// TwinCAT 3 PLC project XMLServerTesten
// ProgramVersion: 3.1.4023.0
// libraries:
//   Tc2_Standard, * (Beckhoff Automation GmbH)
//   Tc2_System, * (Beckhoff Automation GmbH)
//   Tc2_Utilities, * (Beckhoff Automation GmbH)
//   Tc2_XmlDataSrv, * (Beckhoff Automation GmbH)
//   Tc3_Module, * (Beckhoff Automation GmbH)
// project tree:
//   DUTs/ st_Datensatz.TcDUT, ST_TimeDiff.TcDUT (not stored), XMLHeader.TcDUT
//   / PlcTask.TcTTO (not stored)
//   POUs/ Get_Diff.TcPOU, fileT_to_sysT.TcPOU (not stored), MAIN.TcPOU, POU.TcPOU, RecordEndTime.TcPOU, RecordStartTime.TcPOU, write_to_Buffer.TcPOU, write_to_XML.TcPOU, XMLTesten.TcPOU

// ---- DUTs/st_Datensatz.TcDUT
TYPE st_Datensatz :
STRUCT
	Timestamp : STRING ;
	roomnum : REAL;
	temp : REAL;
	signal3 : REAL;
	signal4 : REAL;
	signal5 : REAL;
	signal6 : REAL;
	signal7 : REAL;
	signal8 : REAL;
END_STRUCT
END_TYPE

// ---- DUTs/XMLHeader.TcDUT
TYPE XMLHeader :
STRUCT
	MaschineNummer : STRING:= '1234567890';
	Manufacturer : STRING := 'Beckhoff';
	Maschinetype : STRING:= 'cx2040.1.1.1';
	Customer : STRING:= 'liyizhen23333';
	WriteTimeDiff : ST_TimeDiff;
END_STRUCT
END_TYPE

// ---- POUs/Get_Diff.TcPOU
FUNCTION_BLOCK Get_Diff
VAR_INPUT
	BeginLo: UDINT;
	BeginHi: UDINT;
	EndLo: UDINT;
	EndHi: UDINT;
END_VAR
VAR_OUTPUT
	WriteTimeDiff: ST_TimeDiff;
END_VAR
VAR
	HiDiff : UDINT;
	LoDiff : UDINT;
	SysTime : TIMESTRUCT;
	SysTimeBegin: TIMESTRUCT;
	SysTimeFinish: TIMESTRUCT;
	fileT_to_sysT_Begin: fileT_to_sysT;
	fileT_to_sysT_Finish: fileT_to_sysT;
END_VAR

HiDiff := EndHi - BeginHi;
LoDiff := EndLo - BeginLo;

//change hex time to hh:mm:ss time
fileT_to_sysT_Begin(T_LoDW := LoDiff, T_HiDW := HiDiff);
SysTime := fileT_to_sysT_Begin.sysT;

WriteTimeDiff.mMillisecond:= SysTime.wMilliseconds;
WriteTimeDiff.sSecond:= SysTime.wSecond;

END_FUNCTION_BLOCK

// ---- POUs/MAIN.TcPOU
PROGRAM MAIN
VAR
	XMLTesten : XMLTesten;
END_VAR

XMLTesten();

END_PROGRAM

// ---- POUs/XMLTesten.TcPOU
FUNCTION_BLOCK XMLTesten
VAR_INPUT
END_VAR
VAR_OUTPUT
END_VAR
VAR
	bFinish : BOOL;
	RecordStartTime : RecordStartTime;
	write_to_Buffer : write_to_Buffer;
	RecordEndTime : RecordEndTime;
	write_to_XML : write_to_XML;
	get_Diff : get_Diff;
	
	Buffer : ARRAY[1..100] OF st_Datensatz;
	m: INT :=1;
	StopRecordStart: BOOL := TRUE;
	DownTrigDetect: F_TRIG;
	WriteTimeDiff: ST_TimeDiff;
END_VAR

//record the start timestamp of writing to buffer
IF StopRecordStart THEN
	RecordStartTime(StartFlag := TRUE);
END_IF
StopRecordStart := FALSE; 			//be set so that the start timestamp is not refreshed when writing datensatz2

//when recordstarttime is finished the datensatz is written
IF RecordStartTime.RecordStFinish THEN
	write_to_Buffer(m := m,startrecord := TRUE);
	Buffer[m]:= write_to_Buffer.Datensatz;
	m :=m+1;
END_IF

//when 100 datensatz are written in buffer, record the end timestamp
IF m = 101 THEN
	RecordEndTime(EndFlag := TRUE);
	bFinish :=TRUE;
	m :=102;
END_IF

IF m = 110 THEN
	m := 1;
END_IF

//get timeintervall for writing into buffer (10ms*n)
get_Diff(WriteTimeDiff=>WriteTimeDiff,BeginLo := RecordStartTime.BeginLo,BeginHi := RecordStartTime.BeginHi,EndLo := RecordEndTime.EndLo, EndHi := RecordEndTime.EndHi);

//write data from buffer to xml file
IF bFinish THEN
	write_to_XML(WriteTimeDiffHeader := WriteTimeDiff,LogInput := Buffer,bExecute := TRUE);
END_IF

END_FUNCTION_BLOCK

// ---- POUs/RecordStartTime.TcPOU
FUNCTION_BLOCK RecordStartTime
VAR_INPUT
	StartFlag: BOOL := FALSE;
END_VAR
VAR_OUTPUT
	RecordStFinish : BOOL :=FALSE;
	BeginLo: UDINT;
	BeginHi: UDINT;
END_VAR
VAR
	UpTrigDetect: R_TRIG;
	MyTimer: getsystemtime;
	Delay: TON;
END_VAR

//start to get system time
MyTimer();

//detect the trigger: false to true
UpTrigDetect(CLK:=StartFlag);

//record beginning Timestamp of initializing period
IF UpTrigDetect.Q THEN
	BeginLo := MyTimer.timeLoDW;								
	BeginHi := MyTimer.timeHiDW;
END_IF

RecordStFinish := TRUE;

//time to wait before next cycle

Delay(IN := TRUE, PT := T#5S);            
IF NOT(Delay.Q) THEN
	RETURN;
END_IF
Delay.IN := FALSE;

END_FUNCTION_BLOCK

// ---- POUs/write_to_Buffer.TcPOU
FUNCTION_BLOCK write_to_Buffer
VAR_INPUT
	startrecord : BOOL;
END_VAR
VAR_OUTPUT
	Datensatz : st_Datensatz;
END_VAR
VAR
	GetTime : NT_GetTime;
	GETTIMESTART : BOOL :=TRUE;
	Timestamp : T_Filetime;
	MyTimer: getsystemtime;
	TimestampSYS: TIMESTRUCT;
END_VAR

//100 values in array
	//GetTime(START := GETTIMESTART,TIMESTR => Timestamp);
	//Datensatz.Timestamp := SYSTEMTIME_TO_STRING(Timestamp);
	MyTimer();
	IF startrecord THEN
		Timestamp.dwLowDateTime:= MyTimer.timeLoDW;							
		Timestamp.dwHighDateTime := MyTimer.timeHiDW;
		TimestampSYS := FILETIME_TO_SYSTEMTIME(Timestamp);
		Datensatz.Timestamp := SYSTEMTIME_TO_STRING(TimestampSYS);
	END_IF
	Datensatz.temp := 1.99999;
	Datensatz.roomnum := 0.99999; 	
	Datensatz.signal3 := 20.99999;
	Datensatz.signal4 := 21.99999;
	Datensatz.signal5 := 22.99999;
	Datensatz.signal6 := 23.99999;
	Datensatz.signal7 := 24.99999;
	Datensatz.signal8 := 25.99999;

END_FUNCTION_BLOCK

// ---- POUs/RecordEndTime.TcPOU
FUNCTION_BLOCK RecordEndTime
VAR_INPUT
	EndFlag: BOOL := FALSE;
END_VAR
VAR_OUTPUT
	RecordEndFinish : BOOL :=FALSE;
	EndLo: UDINT;
	EndHi: UDINT;
END_VAR
VAR
	UpTrigDetect: R_TRIG;
	MyTimer: getsystemtime;
END_VAR

//start to get system time
MyTimer();

//detect the trigger: false to true
UpTrigDetect(CLK:=EndFlag);

//record ending Timestamp of initializing period
IF UpTrigDetect.Q THEN
	EndHi := MyTimer.timeHiDW;
	EndLo := MyTimer.timeLoDW;
END_IF
RecordEndFinish :=TRUE;

END_FUNCTION_BLOCK

// ---- POUs/write_to_XML.TcPOU
FUNCTION_BLOCK write_to_XML
VAR_INPUT
	LogInput : ARRAY[1..100] OF st_Datensatz;
	bExecute 		: BOOL := FALSE;
END_VAR
VAR_OUTPUT
	WriteTimeDiff: ST_TimeDiff;
	bBusy : BOOL;
END_VAR
VAR
	bExecuteValue 		: BOOL;
	get_Diff : get_Diff;
	XmlSrvWriteValue : FB_XmlSrvWrite;
  sFilePath 	: T_MaxString := 'C:\temp_Yizhen\Test.xml';  			//disable for CE
  //sFilePath 	: T_MaxString := '\Hard Disk\Test.xml';		//enable for CE
  sXPathData 		: T_MaxString := '/datafromroom/datapart';
  	INPUT: int;
	Error: BOOL;
	ErrID: UDINT;
	MyTimer: getsystemtime;
	UpTrigDetect: R_TRIG;
	DownTrigDetect: F_TRIG;
	fileT_to_sysT_Before: fileT_to_sysT;
	fileT_to_sysT_After: fileT_to_sysT;
	SysTimeBefore: TIMESTRUCT;
	SysTimeAfter: TIMESTRUCT;
	BeginLo: UDINT;
	BeginHi: UDINT;
	EndLo: UDINT;
	EndHi: UDINT;
	MyTimer2: getsystemtime;
	Header: XMLHeader;
	XmlSrvWriteHeader: FB_XmlSrvWrite;
	sXPathHeader: T_MaxString := '/datafromroom/Header';
END_VAR

(* 	Sample1 creates an XML-file under the path C:\Test.xml and writes value1 to it. 
	Existing file will be overwritten.
	FUNCTIONBLOCK: FB_XmlSrvWrite *)
	
//start to get system time	
MyTimer();

//detect the trigger: false to true
UpTrigDetect(CLK:=bExecute);

//detect the trigger: false to true
DownTrigDetect(CLK:=XmlSrvWriteValue.bBusy);

//record beginning Timestamp of writing period
IF UpTrigDetect.Q THEN
	BeginLo := MyTimer.timeLoDW;							
	BeginHi := MyTimer.timeHiDW;
END_IF

//write the xml header
XmlSrvWriteHeader(
	nMode	:= XMLSRV_ADDMISSING, 
  pSymAddr	:= ADR(Header),
  cbSymSize	:= SIZEOF(Header), 
  sFilePath	:= sFilePath,
  sXPath	:= sXPathHeader,
  bExecute	:= bExecute
);

//when xml header is done, start to write the values
IF NOT(XmlSrvWriteHeader.bBusy) THEN
	bExecuteValue := TRUE;
END_IF

//write values to xml file	
XmlSrvWriteValue(
  nMode		:= XMLSRV_ADDMISSING, 
  pSymAddr	:= ADR(LogInput),
  cbSymSize	:= SIZEOF(LogInput), 
  sFilePath	:= sFilePath,
  sXPath	:= sXPathData,
  bExecute	:= bExecuteValue
);

(*Error := XmlSrvWriteValue.bError;
ErrID := XmlSrvWriteValue.nErrId;
bBusy := XmlSrvWriteValue.bBusy; *)

//record ending Timestamp of writing period
IF DownTrigDetect.Q THEN
	EndHi := MyTimer.timeHiDW;
	EndLo := MyTimer.timeLoDW;							
END_IF

//get timeintervall for writing into xml file
get_Diff(BeginLo := BeginLo,BeginHi := BeginHi,EndLo := EndLo, EndHi := EndHi);
WriteTimeDiff:=get_Diff.WriteTimeDiff;

END_FUNCTION_BLOCK

// ---- POUs/POU.TcPOU
FUNCTION_BLOCK POU
VAR_INPUT
END_VAR
VAR_OUTPUT
END_VAR
VAR
END_VAR

// NETWORK 1

END_FUNCTION_BLOCK
